FUNCTION_BLOCK RunUnitCellularAIO EXTENDS RunUnitIndexerMaster
VAR_INPUT
	allHit : BOOL;
	allReach : BOOL;
	allRelease : BOOL;
END_VAR
VAR_OUTPUT
	triggerHit : BOOL;
	triggerRelease : BOOL;
END_VAR
VAR
	ioConveyor : POINTER TO ioBundleConveyor;
	runTimer : TON;
END_VAR
VAR PERSISTENT
	//Checkpoints
	commandTriggerRaise: TIME; //trigger point
	commandReceivingTime : TIME; //if not all lifter done until then , slowdown conveyor motion
END_VAR

//implement state 3
isLastSlotOccupied := TRUE; //always pass carreir even empty material

SUPER^(); //run indexer master

IF bSerialTransition AND State = 1 THEN
	NextState := 16#10; //state override : release lifters
END_IF
IF bSerialTransition AND state=2 THEN
	//moving
	//timer setup and run
	runTimer.IN := TRUE;
	runTimer.PT := commandTriggerRaise;
	ioConveyor^.run := TRUE;

	NextState := 16#11; //re-direct
END_IF

CASE outputState OF
	//-------------------------release lifters
	16#10:
	IF allRelease THEN
		//reset
		triggerRelease:=FALSE;				
		NextState := 2; //wait syncAckowledged 
	END_IF
	//------------------start running
	16#11:
	IF runTimer.Q THEN	
		triggerHit := TRUE;//until trigger raise reached , trigger all lifter to move
		bSerialTransition:= TRUE; //serial transition
		
		runTimer.IN := FALSE;
	ELSE
		//on-going , not trigger lifter
	END_IF
	16#12:
	IF allHit THEN
		triggerHit:=FALSE;
		syncEngaged := FALSE ;// sending over
		bSerialTransition:= TRUE; //serial transition
	ELSIF timeoutTimer.Q THEN
		//sending error , raising alarm
		AlarmCode := eErrorCodes.AC_CONVEYOR_JAMMED;
	END_IF
	16#13:
	IF allReach THEN	
		bSerialTransition := TRUE; //since working signal raised by individual lifter?
	ELSIF timeoutTimer.Q THEN	
		//receiving error , should stop conveyor	
		AlarmCode := eErrorCodes.AC_CONVEYOR_NOT_REACHED;
	END_IF
	16#14:
	IF Upstream<>0 AND_THEN Upstream^.syncEngaged THEN
		//receive data
		SlotBase^.Valid := Upstream^.syncMatValid;
		SlotBase^.Id := Upstream^.syncMatId;
		//After all reached , then pull upstream
		Upstream^.syncAcknowledged := TRUE;//pull upstream when ready
		bSerialTransition:= TRUE; //serial transition	
	ELSIF timeoutTimer.Q THEN 
		//waiting upstream , reminder
	END_IF
	16#15:
	//wait until upstream action done
	bSerialTransition := Upstream<>0 AND_THEN NOT Upstream^.syncEngaged;
	IF bSerialTransition THEN
		//start count-down
		runTimer.PT := commandReceivingTime;
		runTimer.IN := TRUE;
	ELSIF NOT bSerialTransition AND timeoutTimer.Q THEN
		//reminder	
	END_IF
	16#16:
	// on extension , only one oppertunity
	IF runTimer.Q THEN
		runTimer.IN := FALSE;
		ioConveyor^.run := FALSE; //conveyor stopped
		
		triggerRelease:=TRUE;
		Upstream^.syncAcknowledged := FALSE; //inform done
		
		NextState := 0;//done
	ELSE
		//wait motion done	
	END_IF	
	//------------------------end of running
END_CASE
//run timer
runTimer(IN:= , PT:= , Q=> , ET=> );

METHOD ConfigureRead : CellDataBlock
VAR_INPUT
	input : CellDataBlock;
	mode : eModes;
END_VAR
CASE input.unit.config.configId OF 
	0:
		ConfigureRead.unit.config.value := TO_DWORD(commandTriggerRaise);
	1:
		 ConfigureRead.unit.config.value:= TO_DWORD(commandReceivingTime);
	
END_CASE
END_METHOD

METHOD ConfigureWrite : BOOL
VAR_INPUT
	input : CellDataBlock;
	mode : eModes;
END_VAR
CASE input.unit.config.configId OF 
	0:
		commandTriggerRaise := TO_TIME(input.unit.config.value);
	1:
		commandReceivingTime := TO_TIME(input.unit.config.value);
	
END_CASE
END_METHOD

METHOD FB_init : BOOL
VAR_INPUT
	bInitRetains : BOOL; // if TRUE, the retain variables are initialized (warm start / cold start)
	bInCopyCode : BOOL;  // if TRUE, the instance afterwards gets moved into the copy code (online change)
	
	argParent : POINTER TO RunUnitGeneric;
	argSlotBase : POINTER TO RunMaterial;
	argSlotLast : POINTER TO RunMaterial;
	
	argUpstream : POINTER TO RunUnitTransporterBase;
	argAxis : POINTER TO RunAxis;

	argIo : pointer to ioBundleConveyor;
END_VAR
//initialize 
Parent := argParent;
SlotBase := argSlotBase;
SlotLast := argSlotLast;

Axis := 0; //no servo axis
Upstream := argUpstream;

ioConveyor := argIo;
END_METHOD

METHOD Initialize : BOOL
VAR_INPUT
END_VAR
//direct change state
NextState := eSpecialStates.INITIAL_END;
Initialize := SUPER^.Initialize();
END_METHOD

END_FUNCTION_BLOCK

(* stored: Version 1.1.0.1, ProductVersion 3.1.4022.10
   POU RunUnitCellularAIO: Id {b0aa6adc-8e97-4df4-866b-f03dd216654d}, SpecialFunc None
   Method ConfigureRead: Id {05136bdf-c622-49ad-a859-e6a0ec422b6e}
   Method ConfigureWrite: Id {94318e9b-dc61-40e3-b66a-8483f769d4c2}
   Method FB_init: Id {94431706-316d-43bf-8737-4bc97fe6d821}
   Method Initialize: Id {a1a56396-50b5-4a67-b24b-77ca39f7b67a} *)
